(* CODESYS project Modbus_Test_Project_Virtual_RECOVERED_2025-07-04T10-09-00.project

Project tree, tasks and I/O mapping:
  CODESYS_Control_Win_V3 : CODESYS Virtual Control for Linux SL, CODESYS, order no. 2302000005, version 4.16.0.0
    application Application
      libraries: ModbusFB, 4.4.0.0 (CODESYS); Util, 3.5.19.0 (System)
      task Task (cyclic, interval t#20ms, priority 1) calls Main
      function block FB_ModbusSlave [ST]
      program Main [ST]
*)

// CODESYS_Control_Win_V3/Application/Main
PROGRAM Main
VAR
	modbusSlave: FB_ModbusSlave;
END_VAR

modbusSlave();

END_PROGRAM

// CODESYS_Control_Win_V3/Application/FB_ModbusSlave
FUNCTION_BLOCK FB_ModbusSlave
VAR
	aDiscreteInputsMemory: ARRAY[0..9] OF BOOL;
	aCoilsMemory1: ARRAY[0..4] OF BOOL;
	aCoilsMemory2: ARRAY[0..4] OF BOOL;
	aInputRegistersMemory1: ARRAY[0..6] OF UINT;
	aInputRegistersMemory2: ARRAY[0..2] OF UINT;
	aHoldingRegistersMemory: ARRAY[0..6] OF UINT;
END_VAR
VAR CONSTANT
	/// custom defined fcsSupported 
	fcsSupported: ModbusFB.SupportedFcs := (ReadCoils := TRUE, ReadDiscreteInputs := TRUE, ReadHoldingRegisters := TRUE, ReadInputRegisters := TRUE, WriteSingleCoil := TRUE, WriteSingleRegister := TRUE);
	/// Simple multi-section "data model".
	/// This "data model" is completely memory mapped (all "data items" mapped to memory).
	/// It contains non-consecutive "data items" and non-consecutive data item memory to demonstrate how to setup such a configuration.
	/// "plain vanilla" setup can be done also, see "discrete inputs".
	/// "discrete inputs" - "plain vanilla": consecutive "data items" (0..n-1) and consecutive data item memory (one block of memory for all "data items").
	aDiscreteInputsSections: ARRAY[0..0] OF ModbusFB.TableSection := [(uiStart := 0, uiNumDataItems := 10, pStartAddr := ADR(aDiscreteInputsMemory[0]), uiDataItemSize := 8)];
	/// "coils" - consecutive "data items" and non-consecutive data item memory
	aCoilsSections: ARRAY[0..1] OF ModbusFB.TableSection := [(uiStart := 0, uiNumDataItems := 5, pStartAddr := ADR(aCoilsMemory1[0]), uiDataItemSize := 8), (uiStart := 5, uiNumDataItems := 5, pStartAddr := ADR(aCoilsMemory2[0]), uiDataItemSize := 8)];
	/// "input registers" - non-consecutive "data items" and non-consecutive data item memory
	aInputRegistersSections: ARRAY[0..2] OF ModbusFB.TableSection := [(uiStart := 0, uiNumDataItems := 3, pStartAddr := ADR(aInputRegistersMemory1[0]), uiDataItemSize := 16), (uiStart := 5, uiNumDataItems := 4, pStartAddr := ADR(aInputRegistersMemory1[3]), uiDataItemSize := 16), (uiStart := 10, uiNumDataItems := 3, pStartAddr := ADR(aInputRegistersMemory2[0]), uiDataItemSize := 16)];
	/// "holding registers" - consecutive "data items" and consecutive data item memory
	/// "holding registers" 7..9 overlap with "input registers" 10..12
	aHoldingRegistersSections: ARRAY[0..1] OF ModbusFB.TableSection := [(uiStart := 0, uiNumDataItems := 6, pStartAddr := ADR(aHoldingRegistersMemory[0]), uiDataItemSize := 16), (uiStart := 7, uiNumDataItems := 3, pStartAddr := ADR(aInputRegistersMemory2[0]), uiDataItemSize := 16)];
	/// the "data model" tables
	tableDefs: ModbusFB.TableDefinitions := (tableDiscreteInputs := (uiNumSections := 1, pSections := ADR(aDiscreteInputsSections[0])), tableCoils := (uiNumSections := 2, pSections := ADR(aCoilsSections[0])), tableInputRegisters := (uiNumSections := 3, pSections := ADR(aInputRegistersSections[0])), tableHoldingRegisters := (uiNumSections := 2, pSections := ADR(aHoldingRegistersSections[0])));
END_VAR
VAR
	/// our MODBUS TCP server (slave)
	serverTCP: ModbusFB.ServerTCP;
	/// our MODBUS RTU server (slave)
	serverSerial: ModbusFB.ServerSerial;
	initDone: BOOL := FALSE;
END_VAR

IF NOT initDone THEN
	initDone := TRUE;
	// configure tcpServer 
	serverTCP(fcsSupported:=fcsSupported, dataModel:=tableDefs, wsInterfaceName:="", uiPort:=1100);
	// configure serialServer 
END_IF

// call the server FB's
serverTCP(xEnable:=TRUE);
serverSerial(xEnable:=TRUE);

END_FUNCTION_BLOCK
